LIN {X 104.008,Y 270.706,Z 49.708,A -111.017,B 90.000,C 0.000} C_DIS
LIN {X 101.698,Y 271.583,Z 50.088,A -110.529,B 90.000,C 0.000} C_DIS
LIN {X 99.370,Y 272.444,Z 50.382,A -110.039,B 90.000,C 0.000} C_DIS
LIN {X 97.025,Y 273.287,Z 50.577,A -109.546,B 90.000,C 0.000} C_DIS
LIN {X 94.667,Y 274.113,Z 50.659,A -109.053,B 90.000,C 0.000} C_DIS
LIN {X 92.301,Y 274.919,Z 50.616,A -108.559,B 90.000,C 0.000} C_DIS
LIN {X 89.935,Y 275.702,Z 50.429,A -108.066,B 90.000,C 0.000} C_DIS
LIN {X 87.578,Y 276.460,Z 50.081,A -107.577,B 90.000,C 0.000} C_DIS
LIN {X 85.245,Y 277.188,Z 49.557,A -107.095,B 90.000,C 0.000} C_DIS
LIN {X 82.955,Y 277.882,Z 48.835,A -106.622,B 90.000,C 0.000} C_DIS
LIN {X 80.728,Y 278.537,Z 47.907,A -106.163,B 90.000,C 0.000} C_DIS
LIN {X 78.591,Y 279.148,Z 46.763,A -105.724,B 90.000,C 0.000} C_DIS
LIN {X 76.574,Y 279.708,Z 45.397,A -105.310,B 90.000,C 0.000} C_DIS
LIN {X 74.710,Y 280.211,Z 43.809,A -104.929,B 90.000,C 0.000} C_DIS
LIN {X 74.195,Y 278.279,Z 43.809,A -104.929,B 90.000,C 0.000} C_DIS
WAIT SEC 0.1
RET=EKI_SetBool("oxy","torchState",FALSE)
RET = EKI_Send("oxy","torchState")
LIN {X 69.558,Y 260.886,Z 43.809,A -104.929,B 90.000,C 0.000} C_DIS
LIN {X 75.805,Y 259.140,Z 150.506,A -106.306,B 90.000,C 0.000} C_DIS
LIN {X 80.859,Y 276.416,Z 150.506,A -106.306,B 90.000,C 0.000} C_DIS
LIN {X 81.420,Y 278.336,Z 150.506,A -106.306,B 90.000,C 0.000} C_DIS
WAIT SEC 1.75
RET=EKI_SetBool("oxy","torchState",TRUE)
RET = EKI_Send("oxy","torchState")
LIN {X 83.651,Y 277.667,Z 151.416,A -106.766,B 90.000,C 0.000} C_DIS
LIN {X 85.879,Y 276.988,Z 152.322,A -107.226,B 90.000,C 0.000} C_DIS
LIN {X 88.104,Y 276.290,Z 153.223,A -107.687,B 90.000,C 0.000} C_DIS
LIN {X 90.324,Y 275.569,Z 154.116,A -108.148,B 90.000,C 0.000} C_DIS
LIN {X 92.542,Y 274.835,Z 155.005,A -108.609,B 90.000,C 0.000} C_DIS
LIN {X 94.756,Y 274.079,Z 155.887,A -109.072,B 90.000,C 0.000} C_DIS
LIN {X 96.965,Y 273.303,Z 156.762,A -109.534,B 90.000,C 0.000} C_DIS
LIN {X 99.172,Y 272.513,Z 157.632,A -109.997,B 90.000,C 0.000} C_DIS
LIN {X 101.373,Y 271.702,Z 158.493,A -110.461,B 90.000,C 0.000} C_DIS
LIN {X 103.570,Y 270.870,Z 159.348,A -110.925,B 90.000,C 0.000} C_DIS
LIN {X 105.763,Y 270.023,Z 160.196,A -111.389,B 90.000,C 0.000} C_DIS
LIN {X 107.952,Y 269.157,Z 161.038,A -111.854,B 90.000,C 0.000} C_DIS
LIN {X 110.135,Y 268.268,Z 161.870,A -112.320,B 90.000,C 0.000} C_DIS
LIN {X 112.314,Y 267.363,Z 162.695,A -112.786,B 90.000,C 0.000} C_DIS
LIN {X 114.489,Y 266.442,Z 163.514,A -113.253,B 90.000,C 0.000} C_DIS
LIN {X 116.658,Y 265.499,Z 164.323,A -113.720,B 90.000,C 0.000} C_DIS
LIN {X 118.821,Y 264.536,Z 165.124,A -114.188,B 90.000,C 0.000} C_DIS
LIN {X 120.980,Y 263.556,Z 165.917,A -114.657,B 90.000,C 0.000} C_DIS
LIN {X 123.134,Y 262.559,Z 166.702,A -115.125,B 90.000,C 0.000} C_DIS
LIN {X 125.281,Y 261.541,Z 167.477,A -115.595,B 90.000,C 0.000} C_DIS
LIN {X 125.649,Y 261.366,Z 167.610,A -115.675,B 90.000,C 0.000} C_DIS
LIN {X 124.782,Y 259.564,Z 167.610,A -115.675,B 90.000,C 0.000} C_DIS
WAIT SEC 0.1
RET=EKI_SetBool("oxy","torchState",FALSE)
RET = EKI_Send("oxy","torchState")
LIN {X 116.984,Y 243.341,Z 167.610,A -115.675,B 90.000,C 0.000} C_DIS
LIN {X 167.207,Y 211.995,Z 161.609,A -128.264,B 90.000,C 0.000} C_DIS
LIN {X 178.354,Y 226.128,Z 161.609,A -128.264,B 90.000,C 0.000} C_DIS
LIN {X 179.593,Y 227.698,Z 161.609,A -128.264,B 90.000,C 0.000} C_DIS
WAIT SEC 1.75
RET=EKI_SetBool("oxy","torchState",TRUE)
RET = EKI_Send("oxy","torchState")
LIN {X 181.534,Y 226.152,Z 161.910,A -128.754,B 90.000,C 0.000} C_DIS
LIN {X 183.466,Y 224.589,Z 162.178,A -129.245,B 90.000,C 0.000} C_DIS
LIN {X 185.386,Y 223.005,Z 162.409,A -129.737,B 90.000,C 0.000} C_DIS
LIN {X 187.296,Y 221.405,Z 162.606,A -130.229,B 90.000,C 0.000} C_DIS
LIN {X 189.193,Y 219.785,Z 162.765,A -130.722,B 90.000,C 0.000} C_DIS
LIN {X 191.079,Y 218.148,Z 162.891,A -131.215,B 90.000,C 0.000} C_DIS
LIN {X 192.950,Y 216.494,Z 162.978,A -131.709,B 90.000,C 0.000} C_DIS
LIN {X 194.809,Y 214.823,Z 163.033,A -132.203,B 90.000,C 0.000} C_DIS
LIN {X 196.653,Y 213.136,Z 163.049,A -132.697,B 90.000,C 0.000} C_DIS
LIN {X 198.484,Y 211.433,Z 163.032,A -133.191,B 90.000,C 0.000} C_DIS
LIN {X 200.298,Y 209.715,Z 162.976,A -133.684,B 90.000,C 0.000} C_DIS
LIN {X 202.097,Y 207.982,Z 162.887,A -134.178,B 90.000,C 0.000} C_DIS
LIN {X 203.880,Y 206.234,Z 162.759,A -134.671,B 90.000,C 0.000} C_DIS
LIN {X 204.377,Y 205.742,Z 162.719,A -134.809,B 90.000,C 0.000} C_DIS
LIN {X 202.968,Y 204.324,Z 162.719,A -134.809,B 90.000,C 0.000} C_DIS
WAIT SEC 0.1
RET=EKI_SetBool("oxy","torchState",FALSE)
RET = EKI_Send("oxy","torchState")
LIN {X 190.282,Y 191.553,Z 162.719,A -134.809,B 90.000,C 0.000} C_DIS
LIN {X 103.854,Y 249.227,Z 233.497,A -112.622,B 90.000,C 0.000} C_DIS
LIN {X 110.778,Y 265.842,Z 233.497,A -112.622,B 90.000,C 0.000} C_DIS
LIN {X 111.547,Y 267.689,Z 233.497,A -112.622,B 90.000,C 0.000} C_DIS
WAIT SEC 1.75
RET=EKI_SetBool("oxy","torchState",TRUE)
RET = EKI_Send("oxy","torchState")
LIN {X 109.363,Y 268.583,Z 232.674,A -112.155,B 90.000,C 0.000} C_DIS
LIN {X 107.172,Y 269.465,Z 231.856,A -111.689,B 90.000,C 0.000} C_DIS
LIN {X 104.974,Y 270.334,Z 231.043,A -111.222,B 90.000,C 0.000} C_DIS
LIN {X 102.762,Y 271.178,Z 230.240,A -110.754,B 90.000,C 0.000} C_DIS
LIN {X 100.543,Y 272.008,Z 229.442,A -110.286,B 90.000,C 0.000} C_DIS
LIN {X 98.318,Y 272.825,Z 228.650,A -109.818,B 90.000,C 0.000} C_DIS
LIN {X 96.079,Y 273.616,Z 227.867,A -109.349,B 90.000,C 0.000} C_DIS
LIN {X 93.835,Y 274.394,Z 227.090,A -108.879,B 90.000,C 0.000} C_DIS
LIN {X 91.583,Y 275.159,Z 226.317,A -108.409,B 90.000,C 0.000} C_DIS
LIN {X 89.320,Y 275.897,Z 225.555,A -107.939,B 90.000,C 0.000} C_DIS
LIN {X 87.051,Y 276.621,Z 224.798,A -107.468,B 90.000,C 0.000} C_DIS
LIN {X 84.775,Y 277.332,Z 224.046,A -106.997,B 90.000,C 0.000} C_DIS
LIN {X 82.488,Y 278.016,Z 223.304,A -106.526,B 90.000,C 0.000} C_DIS
LIN {X 80.195,Y 278.686,Z 222.567,A -106.054,B 90.000,C 0.000} C_DIS
LIN {X 77.897,Y 279.342,Z 221.835,A -105.582,B 90.000,C 0.000} C_DIS
LIN {X 75.588,Y 279.971,Z 221.114,A -105.109,B 90.000,C 0.000} C_DIS
LIN {X 74.122,Y 280.367,Z 220.657,A -104.809,B 90.000,C 0.000} C_DIS
LIN {X 73.611,Y 278.434,Z 220.657,A -104.809,B 90.000,C 0.000} C_DIS
WAIT SEC 0.1
RET=EKI_SetBool("oxy","torchState",FALSE)
RET = EKI_Send("oxy","torchState")
LIN {X 69.010,Y 261.032,Z 220.657,A -104.809,B 90.000,C 0.000} C_DIS
LIN {X -64.526,Y 262.176,Z 229.899,A -76.173,B 90.000,C 0.000} C_DIS
LIN {X -68.828,Y 279.655,Z 229.899,A -76.173,B 90.000,C 0.000} C_DIS
LIN {X -69.306,Y 281.597,Z 229.899,A -76.173,B 90.000,C 0.000} C_DIS
WAIT SEC 1.75
RET=EKI_SetBool("oxy","torchState",TRUE)
RET = EKI_Send("oxy","torchState")
LIN {X -71.691,Y 280.998,Z 229.451,A -75.688,B 90.000,C 0.000} C_DIS
LIN {X -74.076,Y 280.379,Z 229.030,A -75.201,B 90.000,C 0.000} C_DIS
LIN {X -76.460,Y 279.739,Z 228.638,A -74.713,B 90.000,C 0.000} C_DIS
LIN {X -78.843,Y 279.075,Z 228.276,A -74.224,B 90.000,C 0.000} C_DIS
LIN {X -81.224,Y 278.392,Z 227.942,A -73.735,B 90.000,C 0.000} C_DIS
LIN {X -83.603,Y 277.687,Z 227.637,A -73.245,B 90.000,C 0.000} C_DIS
LIN {X -85.979,Y 276.960,Z 227.363,A -72.754,B 90.000,C 0.000} C_DIS
LIN {X -88.351,Y 276.213,Z 227.117,A -72.262,B 90.000,C 0.000} C_DIS
LIN {X -90.720,Y 275.444,Z 226.901,A -71.770,B 90.000,C 0.000} C_DIS
LIN {X -93.084,Y 274.653,Z 226.714,A -71.278,B 90.000,C 0.000} C_DIS
LIN {X -95.141,Y 273.949,Z 226.574,A -70.848,B 90.000,C 0.000} C_DIS
LIN {X -94.484,Y 272.060,Z 226.574,A -70.848,B 90.000,C 0.000} C_DIS
WAIT SEC 0.1
RET=EKI_SetBool("oxy","torchState",FALSE)
RET = EKI_Send("oxy","torchState")
LIN {X -88.579,Y 255.056,Z 226.574,A -70.848,B 90.000,C 0.000} C_DIS
LIN {X -121.741,Y 240.996,Z 227.857,A -63.199,B 90.000,C 0.000} C_DIS
LIN {X -129.857,Y 257.063,Z 227.857,A -63.199,B 90.000,C 0.000} C_DIS
LIN {X -130.759,Y 258.848,Z 227.857,A -63.199,B 90.000,C 0.000} C_DIS
WAIT SEC 1.75
RET=EKI_SetBool("oxy","torchState",TRUE)
RET = EKI_Send("oxy","torchState")
LIN {X -132.966,Y 257.720,Z 228.184,A -62.709,B 90.000,C 0.000} C_DIS
LIN {X -135.160,Y 256.576,Z 228.537,A -62.220,B 90.000,C 0.000} C_DIS
LIN {X -137.341,Y 255.416,Z 228.919,A -61.732,B 90.000,C 0.000} C_DIS
LIN {X -139.507,Y 254.238,Z 229.332,A -61.245,B 90.000,C 0.000} C_DIS
LIN {X -141.659,Y 253.046,Z 229.772,A -60.759,B 90.000,C 0.000} C_DIS
LIN {X -143.797,Y 251.837,Z 230.241,A -60.274,B 90.000,C 0.000} C_DIS
LIN {X -145.918,Y 250.613,Z 230.740,A -59.790,B 90.000,C 0.000} C_DIS
LIN {X -148.025,Y 249.375,Z 231.266,A -59.307,B 90.000,C 0.000} C_DIS
LIN {X -150.116,Y 248.122,Z 231.822,A -58.826,B 90.000,C 0.000} C_DIS
LIN {X -152.190,Y 246.855,Z 232.408,A -58.346,B 90.000,C 0.000} C_DIS
LIN {X -154.248,Y 245.576,Z 233.019,A -57.867,B 90.000,C 0.000} C_DIS
LIN {X -156.288,Y 244.282,Z 233.662,A -57.389,B 90.000,C 0.000} C_DIS
LIN {X -158.311,Y 242.975,Z 234.333,A -56.914,B 90.000,C 0.000} C_DIS
LIN {X -160.317,Y 241.658,Z 235.030,A -56.439,B 90.000,C 0.000} C_DIS
LIN {X -162.304,Y 240.327,Z 235.759,A -55.967,B 90.000,C 0.000} C_DIS
LIN {X -163.327,Y 239.633,Z 236.145,A -55.723,B 90.000,C 0.000} C_DIS
LIN {X -162.201,Y 237.981,Z 236.145,A -55.723,B 90.000,C 0.000} C_DIS
WAIT SEC 0.1
RET=EKI_SetBool("oxy","torchState",FALSE)
RET = EKI_Send("oxy","torchState")
LIN {X -152.063,Y 223.107,Z 236.145,A -55.723,B 90.000,C 0.000} C_DIS
LIN {X -193.754,Y 188.041,Z 184.833,A -44.143,B 90.000,C 0.000} C_DIS
LIN {X -206.671,Y 200.577,Z 184.833,A -44.143,B 90.000,C 0.000} C_DIS
LIN {X -208.106,Y 201.970,Z 184.833,A -44.143,B 90.000,C 0.000} C_DIS
WAIT SEC 1.75
RET=EKI_SetBool("oxy","torchState",TRUE)
RET = EKI_Send("oxy","torchState")
LIN {X -209.836,Y 200.170,Z 184.973,A -43.650,B 90.000,C 0.000} C_DIS
LIN {X -211.551,Y 198.358,Z 185.125,A -43.157,B 90.000,C 0.000} C_DIS
LIN {X -213.249,Y 196.530,Z 185.278,A -42.664,B 90.000,C 0.000} C_DIS
LIN {X -214.932,Y 194.688,Z 185.421,A -42.171,B 90.000,C 0.000} C_DIS
LIN {X -216.601,Y 192.831,Z 185.547,A -41.677,B 90.000,C 0.000} C_DIS
LIN {X -218.254,Y 190.958,Z 185.639,A -41.184,B 90.000,C 0.000} C_DIS
LIN {X -219.891,Y 189.070,Z 185.690,A -40.690,B 90.000,C 0.000} C_DIS
LIN {X -221.513,Y 187.167,Z 185.690,A -40.196,B 90.000,C 0.000} C_DIS
LIN {X -223.118,Y 185.252,Z 185.626,A -39.702,B 90.000,C 0.000} C_DIS
LIN {X -223.243,Y 185.101,Z 185.618,A -39.664,B 90.000,C 0.000} C_DIS
LIN {X -221.703,Y 183.825,Z 185.618,A -39.664,B 90.000,C 0.000} C_DIS
WAIT SEC 0.1
RET=EKI_SetBool("oxy","torchState",FALSE)
RET = EKI_Send("oxy","torchState")
LIN {X -207.847,Y 172.336,Z 185.618,A -39.664,B 90.000,C 0.000} C_DIS
LIN {X -156.294,Y 220.164,Z 47.437,A -54.629,B 90.000,C 0.000} C_DIS
LIN {X -166.714,Y 234.841,Z 47.437,A -54.629,B 90.000,C 0.000} C_DIS
LIN {X -167.872,Y 236.472,Z 47.437,A -54.629,B 90.000,C 0.000} C_DIS
WAIT SEC 1.75
RET=EKI_SetBool("oxy","torchState",TRUE)
RET = EKI_Send("oxy","torchState")
LIN {X -165.844,Y 237.898,Z 47.759,A -55.119,B 90.000,C 0.000} C_DIS
LIN {X -163.810,Y 239.303,Z 48.131,A -55.607,B 90.000,C 0.000} C_DIS
LIN {X -161.771,Y 240.686,Z 48.554,A -56.094,B 90.000,C 0.000} C_DIS
LIN {X -159.728,Y 242.046,Z 49.027,A -56.579,B 90.000,C 0.000} C_DIS
LIN {X -157.682,Y 243.384,Z 49.551,A -57.062,B 90.000,C 0.000} C_DIS
LIN {X -155.635,Y 244.699,Z 50.126,A -57.542,B 90.000,C 0.000} C_DIS
LIN {X -153.588,Y 245.989,Z 50.752,A -58.021,B 90.000,C 0.000} C_DIS
LIN {X -151.541,Y 247.256,Z 51.424,A -58.496,B 90.000,C 0.000} C_DIS
LIN {X -149.491,Y 248.500,Z 52.131,A -58.970,B 90.000,C 0.000} C_DIS
LIN {X -147.436,Y 249.723,Z 52.859,A -59.442,B 90.000,C 0.000} C_DIS
LIN {X -145.373,Y 250.925,Z 53.598,A -59.914,B 90.000,C 0.000} C_DIS
LIN {X -143.303,Y 252.117,Z 54.335,A -60.386,B 90.000,C 0.000} C_DIS
LIN {X -141.220,Y 253.291,Z 55.062,A -60.859,B 90.000,C 0.000} C_DIS
LIN {X -139.120,Y 254.451,Z 55.766,A -61.333,B 90.000,C 0.000} C_DIS
LIN {X -137.002,Y 255.598,Z 56.434,A -61.808,B 90.000,C 0.000} C_DIS
LIN {X -134.863,Y 256.733,Z 57.055,A -62.287,B 90.000,C 0.000} C_DIS
LIN {X -132.702,Y 257.857,Z 57.618,A -62.768,B 90.000,C 0.000} C_DIS
LIN {X -132.561,Y 257.929,Z 57.653,A -62.799,B 90.000,C 0.000} C_DIS
LIN {X -131.647,Y 256.151,Z 57.653,A -62.799,B 90.000,C 0.000} C_DIS
WAIT SEC 0.1
RET=EKI_SetBool("oxy","torchState",FALSE)
RET = EKI_Send("oxy","torchState")
LIN {X -109.706,Y 213.459,Z 57.653,A -62.799,B 90.000,C 0.000} C_DIS
PTP {A1 0.0,A2 -100.0,A3 150.0,A4 0.0,A5 -50.0,A6 0.0}


END
